// TIA Portal V19 export
DATA_BLOCK "MODE SELECTION DB"   // DB1
{ S7_Optimized_Access := 'FALSE' }
   VAR
      MGF : Struct
         AUTO : Bool;
         MANUAL : Bool;
         STANDBY : Bool;
         "MODE BUFF" : Int;
         "PROCESS BUFF" : Int;
         START : Bool;
         STOP : Bool;
      END_STRUCT;
      UF : Struct
         AUTO : Bool;
         MANUAL : Bool;
         STANDBY : Bool;
         START : Bool;
         STOP : Bool;
      END_STRUCT;
      "UF PLC_1 MODE BUFF" : Int;
      "UF PLC_1 PROCESS BUFF" : Int;
      "DM FEED PUMP" : Struct
         AUTO : Bool;
         MANUAL : Bool;
         STANDBY : Bool;
         "MODE BUFF" : Int;
         "PROCESS BUFF" : Int;
         START : Bool;
         STOP : Bool;
      END_STRUCT;
      "BACK WASH" : Struct
         AUTO : Bool;
         MANUAL : Bool;
         STANDBY : Bool;
         "MODE BUFF" : Int;
         "PROCESS BUFF" : Int;
         START : Bool;
         STOP : Bool;
      END_STRUCT;
   END_VAR
BEGIN
END_DATA_BLOCK
